PROGRAM MAIN
VAR
    diKapSensor1 AT %I* : BOOL ;

    bMinneKapSensor1 : BOOL := 0;
	    diKapSensor2 AT %I* : BOOL ;

    bMinneKapSensor2 : BOOL := 0;
END_VAR

bMinneKapSensor1 := diKapSensor1;
bMinneKapSensor2 := diKapSensor2;

END_PROGRAM

(* stored: Version 1.1.0.1, ProductVersion 3.1.4024.9
   POU MAIN: Id {e94009b9-63c2-4061-8765-e6c01e22484b}, SpecialFunc None *)
